Yaskawa INFORM job: COOLGAS.JBI

/JOB
//NAME COOLGAS
//POS
///NPOS 0,0,0,0,0,0
//INST
///DATE 2015/09/29 10:17
///ATTR SC,RW,MC
///LVARS 10,5,0,0,0,0,0,0
NOP
GETARG LB000 IARG#(1)
SET LI000 LB000
MUL LI000 100
DOUT OT#(18) ON
DOUT OT#(19) OFF
DOUT OT#(51) ON
TIMER T=LI000
DOUT OT#(51) OFF
DOUT OT#(18) OFF
DOUT OT#(19) ON
PULSE OT#(51) T=2.00
END
